(* IEC 61131-3 sources: std_i2980_v2.06_cp053/Source/IMM/ieccontrol/ODC1 (part 7) *)

         IF bGoToEndIf THEN
            aGoToEndIf(iColumn := i);
         ELSIF bGoToBeginLoop THEN
            bGoToBeginLoop := FALSE;
            aGoToBeginLoop(iColumn := i, iInstance := sv_ODCSequenceInt[i][iRow].iCount);
         ELSIF bGoToEndLoop THEN
            bGoToEndLoop := FALSE;
            aGoToEndLoop(iColumn := i, iInstance := sv_ODCSequenceInt[i][iRow].iCount);
         ELSE
            aIncreaseRow(iColumn := i, iEndRow := miEndRow);
         END_IF;
      END_IF;
   END_IF; //odcParallelInfo[i].bColumnActive
END_FOR;

//interesting for HMI to see state of the interpreter
sv_InterpreterParallelInfo := odcParallelInfo;

@END_Body

@@@BEG_Comment@@@
@TL(6)
Interpret the 2 dimensional ODC array.
(Responsible for auto cycle and combined movements)

This needs to be called cyclically until aStatus.bActive = FALSE
This can happen when the interpreter has reached the end of the array/sequence
or when a error happens during interpreting.
@@@END_Comment@@@

@BEG_Body
@TL(84)
(**************************************** WARNING ********************************************
 *** The KEBA Kemro K2 System including software is not intended for safety control tasks! ***
 ***                       For further information see Comment tab!                        ***
 *********************************************************************************************)

bFound := FALSE;
StepPos.iColumn := 0;
StepPos.iRow := 0;

FOR iTmpRow := SearchStartPos.iRow TO sv_iUsedRows DO

   IF iTmpRow = SearchStartPos.iRow THEN
      //start searching in the given column
      iSearchColumn := SearchStartPos.iColumn;
   ELSE
      //start searching in the first column
      iSearchColumn := 1;
   END_IF;

   FOR iTmpColumn := iSearchColumn TO sv_iUsedColumns DO
      IF sv_ODCSequence[iTmpColumn][iTmpRow].iCompId = DeviceId.CompId AND
         INT_TO_DINT(sv_ODCSequence[iTmpColumn][iTmpRow].iIndexId) = DeviceId.IndexId THEN
         IF sv_ODCSequence[iTmpColumn][iTmpRow].iMoveId = MoveId AND
            sv_ODCSequence[iTmpColumn][iTmpRow].iMoveDir = MoveDir AND
            (IntermediateCond = 0 OR // do not care about intermediate condion if we don't search for it?
                                     // FIXME check flag in MoveData instead??
             INT_TO_DINT(sv_ODCSequence[iTmpColumn][iTmpRow].iCount) = IntermediateCond) THEN
            fbDebugTrace2(nODCInterpreter, CONCAT('found exact match of MoveId ',
                                                  DINT_TO_STRING(DeviceId.CompId),
                                                  '.',
                                                  DINT_TO_STRING(DeviceId.IndexId),
                                                  ' ',
                                                  DINT_TO_STRING(MoveId),
                                                  '/',
                                                  DINT_TO_STRING(MoveDir),
                                                  ' ',
                                                  DINT_TO_STRING(IntermediateCond),
                                                  ' at pos:',
                                                  DINT_TO_STRING(iTmpRow),
                                                  '/',
                                                  DINT_TO_STRING(iTmpColumn)));

            StepPos.iColumn := iTmpColumn;
            StepPos.iRow := iTmpRow;
            bFound := TRUE;
            RETURN;

         ELSIF bAllowNonMatchingId AND sv_ODCSequence[iTmpColumn][iTmpRow].iMoveDir = MoveDir THEN
            fbDebugTrace2(nODCInterpreter, CONCAT('found NON exact match of MoveId ',
                                                  DINT_TO_STRING(DeviceId.CompId),
                                                  '.',
                                                  DINT_TO_STRING(DeviceId.IndexId),
                                                  ' ',
                                                  DINT_TO_STRING(MoveId),
                                                  '/',
                                                  DINT_TO_STRING(MoveDir),
                                                  ' ',
                                                  DINT_TO_STRING(IntermediateCond),
                                                  ' at pos:',
                                                  DINT_TO_STRING(iTmpRow),
                                                  '/',
                                                  DINT_TO_STRING(iTmpColumn)));
            StepPos.iColumn := iTmpColumn;
            StepPos.iRow := iTmpRow;
            bFound := TRUE;
         END_IF;
      END_IF;
   END_FOR;
END_FOR;

IF NOT bFound THEN
   fbDebugTrace2(nODCInterpreter, CONCAT('movement ',
                                          DINT_TO_STRING(DeviceId.CompId),
                                          '.',
                                          DINT_TO_STRING(DeviceId.IndexId),
                                          ' ',
                                          DINT_TO_STRING(MoveId),
                                          '/',
                                          DINT_TO_STRING(MoveDir),
                                          ' ',
                                          DINT_TO_STRING(IntermediateCond),
                                          ' not found in auto cycle'));
END_IF;

@END_Body

@@@BEG_Comment@@@
@TL(10)
Search a Movement in the ODC array by DeviceId, MoveId and MovedDir
and return the position in the array.

If bAllowNonMatchingId is TRUE only DeviceId and MoveDir need to match.
But it still tries to get the best match(MoveId equals)

If IntermediateCond is <> 0, it is also checked against iCount when checking for exact match.

When a movement is found bFound is TRUE and StepPos contains the position
of the movement in the ODC array
@@@END_Comment@@@

@BEG_Body
@TL(18)
(**************************************** WARNING ********************************************
 *** The KEBA Kemro K2 System including software is not intended for safety control tasks! ***
 ***                       For further information see Comment tab!                        ***
 *********************************************************************************************)

IF mbFatalError THEN
   mbFatalError := FALSE;

   (* unlock all movements locked by aStopInterpreterInternal *)
   DeviceIdAll.CompId := cCompAll;
   DeviceIdAll.IndexId := cAllDevIndex;

   fbLockUnlock(DeviceId := DeviceIdAll,
               MoveDir  := cMoveAll,
               MoveId   := cMoveAll,
               Mode     := nUnlock);
END_IF;

@END_Body

@@@BEG_Comment@@@
@TL(2)
Notify the Interpreter that the array has been reinitialized
(this clears the fatal error flag)
@@@END_Comment@@@

@BEG_Body
@TL(9)
(**************************************** WARNING ********************************************
 *** The KEBA Kemro K2 System including software is not intended for safety control tasks! ***
 ***                       For further information see Comment tab!                        ***
 *********************************************************************************************)

bError := mbFatalError OR mbNormalError;
bFinished := mbFinished;
bActive := mbActive;

@END_Body

@@@BEG_Comment@@@
@TL(1)
Actual status of the interpreter.
@@@END_Comment@@@

@BEG_Body
@TL(41)
(**************************************** WARNING ********************************************
 *** The KEBA Kemro K2 System including software is not intended for safety control tasks! ***
 ***                       For further information see Comment tab!                        ***
 *********************************************************************************************)

mbStepMode := TRUE;

//stop started movements
StartedMovements := sv_StartedManualMovements;
FOR i := 1 TO StartedMovements.iStartedMovements DO

   //get move number
   fbGetMoveNumber(DeviceId := StartedMovements.MoveData[i].DeviceId,
                   MoveId := StartedMovements.MoveData[i].MoveId,
                   MoveDir := StartedMovements.MoveData[i].MoveDir,
                   iMoveNumber => iMoveNr);

   IF NOT sv_MovementsAvailable[iMoveNr].pMovementData^.bFinishAtInterrupt THEN
      //stop movement
      fbStop(DeviceId := StartedMovements.MoveData[i].DeviceId);
   ELSE
      //movement should finish
      //increase number of active row because otherwise this movement is started
      //again when stepping fwd
      aIncreaseRow(iColumn := StartedMovements.MoveData[i].StepPos.iColumn,
                   iEndRow := miEndRow);
   END_IF;

END_FOR;

//disable steps
FOR i := 1 TO cMaxParallelMovements DO
   IF odcParallelInfo[i].bColumnActive THEN
      odcParallelInfo[i].bDisabled := TRUE;
   END_IF;
END_FOR;

mbActive := FALSE;

sv_InterpreterParallelInfo := odcParallelInfo;

@END_Body

@@@BEG_Comment@@@
@TL(0)

@@@END_Comment@@@

@BEG_Body
@TL(24)
(**************************************** WARNING ********************************************
 *** The KEBA Kemro K2 System including software is not intended for safety control tasks! ***
 ***                       For further information see Comment tab!                        ***
 *********************************************************************************************)

//reset relevant flags
FOR i := 1 TO cMaxParallelMovements DO
   IF odcParallelInfo[i].bColumnActive THEN
      odcParallelInfo[i].bStartSent := FALSE;
      odcParallelInfo[i].bStartConditionWarnPrinted := FALSE;
      odcParallelInfo[i].bActivatedChecked := FALSE;
      odcParallelInfo[i].bDisabled := FALSE;

      //set step state to "active"
      fbSetStepState.StepPos.iColumn := i;
      fbSetStepState.StepPos.iRow := odcParallelInfo[i].iRow;
      fbSetStepState(StepState := nStateActive);
   END_IF;

END_FOR;

mbActive := TRUE;
mbStepMode := FALSE;

@END_Body

@@@BEG_Comment@@@
@TL(0)

@@@END_Comment@@@

@BEG_Body
@TL(23)
(**************************************** WARNING ********************************************
 *** The KEBA Kemro K2 System including software is not intended for safety control tasks! ***
 ***                       For further information see Comment tab!                        ***
 *********************************************************************************************)

//enable steps
FOR i := 1 TO cMaxParallelMovements DO
   IF odcParallelInfo[i].bColumnActive THEN
      odcParallelInfo[i].bDisabled := FALSE;
      odcParallelInfo[i].bStartSent := FALSE;
      odcParallelInfo[i].bStartConditionWarnPrinted := FALSE;
      odcParallelInfo[i].bActivatedChecked := FALSE;

      //set step state to "active"
      fbSetStepState.StepPos.iColumn := i;
      fbSetStepState.StepPos.iRow := odcParallelInfo[i].iRow;
      fbSetStepState(StepState := nStateActive);
   END_IF;

END_FOR;

mbActive := TRUE;

@END_Body

@@@BEG_Comment@@@
@TL(0)

@@@END_Comment@@@

@BEG_Body
@TL(7)
(**************************************** WARNING ********************************************
 *** The KEBA Kemro K2 System including software is not intended for safety control tasks! ***
 ***                       For further information see Comment tab!                        ***
 *********************************************************************************************)

mbStepMode := FALSE;

@END_Body

@@@BEG_Comment@@@
@TL(0)

@@@END_Comment@@@

@BEG_Body
@TL(144)
(**************************************** WARNING ********************************************
 *** The KEBA Kemro K2 System including software is not intended for safety control tasks! ***
 ***                       For further information see Comment tab!                        ***
 *********************************************************************************************)

IF bStartInActualLine THEN
   iStartRow := odcParallelInfo[iColumn].iRow;
ELSE
   iStartRow := (odcParallelInfo[iColumn].iRow - 1);
END_IF;

//reset step state of actually active step
fbSetStepState.StepPos.iColumn := iColumn;
fbSetStepState.StepPos.iRow := odcParallelInfo[iColumn].iRow;
fbSetStepState(StepState := nStateDefault);

iNewActivatedColumn := 0;

//get next line with a "real" movement
FOR iTmpLine := iStartRow TO iEndRow BY -1 DO
   fbDebugTrace2(nODCInterpreter, CONCAT('decreasing IP of column ', DINT_TO_STRING(iColumn),
                                         ' to ', DINT_TO_STRING(iTmpLine)));

   iMoveId := sv_ODCSequence[iColumn][iTmpLine].iMoveId;

   IF (iMoveId = cMoveEndIf) THEN
      // end_if => check if this "if" instance is active or already completely executed
      iCount := sv_ODCSequence[iColumn][iTmpLine].iCount;
      IF (mIFConditionHelpData[iCount].iInternalCount < 2) THEN
         //if or else tree is active
         //set active line in this column to begin of this "if" or "else"
         //so that stepping bwd can continue before this "if / else"
         FOR iLine := (iTmpLine - 1) TO 1 BY -1 DO
            IF ((sv_ODCSequence[iColumn][iLine].iMoveId = cMoveIf) OR (sv_ODCSequence[iColumn][iLine].iMoveId = cMoveElse)) AND
               (sv_ODCSequence[iColumn][iLine].iCount = iCount) THEN
               odcParallelInfo[iColumn].iRow := (iLine - 1);  //set row to "start parallel" step
               EXIT;
            END_IF;
         END_FOR;
         mIFConditionHelpData[iCount].iInternalCount := (mIFConditionHelpData[iCount].iInternalCount - 1);
      ELSE
         //condition completely executed -> do not allow stepping into
         odcParallelInfo[iColumn].iRow := (iTmpLine + 1); //set row to "end parallel" step
         odcParallelInfo[iColumn].bDisabled := TRUE;
         SET_ALARM(Name := erNoStepBwdIntoCondition);
      END_IF;

      EXIT;
   ELSIF (iMoveId = cMoveEndLoop) THEN
      // end loop => stop stepping bwd here
      odcParallelInfo[iColumn].iRow := iTmpLine; //set row to "end loop" step
      odcParallelInfo[iColumn].bDisabled := TRUE;
      SET_ALARM(Name := erNoStepBwdIntoLoop);
      EXIT;
   ELSIF (iMoveId = cMoveBeginLoop) THEN
      // begin of loop => stop stepping bwd here (do not modify line number)
      odcParallelInfo[iColumn].bDisabled := TRUE;
      SET_ALARM(Name := erNoStepBwdOutOfLoop);
      EXIT;
   ELSIF (iMoveId = cMoveBeginSequence) OR (iMoveId = cMoveEndSequence) THEN
      ; // begin or end sequence
   ELSIF (iMoveId = cMoveNone) OR (iMoveId = cMoveBeginGroup) OR (iMoveId = cMoveEndGroup) THEN
      ; //empty step or begin group / end group
   ELSIF (iMoveId = cMoveIf) OR (iMoveId = cMoveElse) THEN
      ; //if , else
   ELSIF iMoveId = cMoveEndParallelOpen THEN
      ; //no special action necessary
   ELSIF iMoveId = cMoveEndParallel THEN
      //get according column and activate it
      FOR iTmpColumn := (iColumn + 1) TO sv_iUsedColumns DO
         IF sv_ODCSequence[iTmpColumn][iTmpLine].iMoveId = cMoveEndParallel THEN
            odcParallelInfo[iTmpColumn].bColumnActive := TRUE;
            odcParallelInfo[iTmpColumn].iRow := (iTmpLine + 1); //necessary to handle more end parallel in one line
            odcParallelInfo[iTmpColumn].bDisabled := TRUE;
            iNewActivatedColumn := iTmpColumn;
            EXIT;
         END_IF;
      END_FOR;
   ELSIF (iMoveId = cMoveStartParallel) OR (iMoveId = cMoveStartParallelOpen) THEN
      bContinueDecreasing := FALSE;
      FOR iTmpColumn := 1 TO sv_iUsedColumns DO
         IF (sv_ODCSequence[iTmpColumn][iTmpLine].iMoveId = cMoveStartParallel) OR
            (sv_ODCSequence[iTmpColumn][iTmpLine].iMoveId = cMoveStartParallelOpen) THEN

            //start parallel or start parallel open found
            IF iTmpColumn < iColumn THEN
               //SP left to actual column found
               //-> deactivate actual column and set line number
               odcParallelInfo[iColumn].iRow := iTmpLine;
               odcParallelInfo[iColumn].bDisabled := FALSE;
               odcParallelInfo[iColumn].bColumnActive := FALSE;
               IF sv_TraceLevel.bODCInterpreter THEN
                  dummy := Print('aDecreaseRow: deactivate column %d ',iColumn);
               END_IF;
            ELSE
               //SP is the most left one in this line
               //-> all SP to the right must be deactivated and their active row must be equal
               bOk := TRUE;
               FOR x := (iTmpColumn + 1) TO sv_iUsedColumns DO
                  //only consider SP entries
                  IF (sv_ODCSequence[x][iTmpLine].iMoveId = cMoveStartParallel) OR
                     (sv_ODCSequence[x][iTmpLine].iMoveId = cMoveStartParallelOpen) THEN
                     bParallelTreeReady := NOT odcParallelInfo[x].bColumnActive AND (odcParallelInfo[x].iRow = iTmpLine);
                     bOk := bOk AND bParallelTreeReady;
                  END_IF;
               END_FOR;

               IF bOk THEN
                  //all parallel trees ready -> decrease line of this column so that it can continue
                  bContinueDecreasing := TRUE;
               ELSE
                  //column still active -> wait in this line
                  odcParallelInfo[iColumn].iRow := iTmpLine;
                  odcParallelInfo[iColumn].bDisabled := TRUE;
                  bContinueDecreasing := FALSE;
               END_IF;
            END_IF;

            EXIT; //exit inner loop
         END_IF;
      END_FOR;

      IF NOT bContinueDecreasing THEN
         EXIT;  // exit outer loop
      END_IF;
   ELSE
      //valid step found -> set line number and disable this step
      IF sv_TraceLevel.bODCInterpreter THEN
         dummy := Print('///////// set active row of column %d to %d ////////////',iColumn, iTmpLine);
      END_IF;
      odcParallelInfo[iColumn].iRow := iTmpLine;
      odcParallelInfo[iColumn].bDisabled := TRUE;
      EXIT;
   END_IF;
END_FOR;

odcParallelInfo[iColumn].bStartSent := FALSE;
odcParallelInfo[iColumn].bStartConditionWarnPrinted := FALSE;
odcParallelInfo[iColumn].bActivatedChecked := FALSE;
odcParallelInfo[iColumn].bPosReachedArrayLinked := FALSE;
odcParallelInfo[iColumn].bMovementReadyArrayLinked := FALSE;

sv_InterpreterParallelInfo[iColumn] := odcParallelInfo[iColumn];

@END_Body

@@@BEG_Comment@@@
@TL(0)

@@@END_Comment@@@
@END_Body

@END_Contents
@@@BEG_Password@@@
NGhzZm9kYzQ=
@@@END_Password@@@

(* ---- ABLogger.pu ---- *)
(*
@h    ! WARNING !
@h    The Kemro K2 system (including software) only meets category B according to EN 954-1,
@h    thus it is not intended for usage in safety-relevant control applications in the field
@h    of personal safety (e.g. emergency stop).
@h    To implement potentially necessary safety-relevant control tasks, always use additional
@h    external safety devices that are intended for the particular purpose, and meet the necessary
@h    functional safety.
@h    For further information see EN 954-1 (EN ISO 13849-1) and/or the K2-x00 user manual, chapter
@h    "CE conformity, directives and standards".

algorithm block for debug purpose, can be used to log single trace lines to file
*)

IMPORT_OVER_LISTFILE
 KFILE_Open_Data
, KFILE_Status

END_IMPORT

ALGORITHM_BLOCK ABLogger #DUMMY_EDIT_BLOCK

VAR
 iResult : DINT (* transferred bytes, return value of KFILE_Read/Write *);
 sTraceString : STRING(255) (* local output trace string *);
END_VAR

ALGORITHM aWriteLine

VAR_INPUT
 sFileName : STRING(255) (* absolute file path *);
 bAppend : BOOL (* append log file *);
END_VAR

VAR_IN_OUT
 sText : STRING(255) (* trace string to log *);
END_VAR

VAR_TEMP
 FileOpenData : KFILE_Open_Data (* file open information *);
 FileStatus : KFILE_Status (* file state *);
 sNewline : STRING(2) := '$n';
 iLen : DINT;
END_VAR
#BEGIN_EDIT_BLOCK
IF (bAppend) THEN
   FileOpenData := KFILE_Open(Name := sFileName,
                              Mode := KFILE_Mode_AppendCreate);
ELSE
   FileOpenData := KFILE_Open(Name := sFileName,
                              Mode := KFILE_Mode_ReadWriteDelete);
END_IF;

IF (FileOpenData.Status = KFILE_Status_OK) THEN
   iLen := LEN(sText);
   IF iLen > 0 THEN
      // write data
      iResult := KFILE_Write(Token := FileOpenData.Token,
                             Length := iLen,
                             Buffer := sText);
   END_IF;
   // CR/LF
   iResult := KFILE_Write(Token := FileOpenData.Token,
                        Length := 2,
                        Buffer := sNewline);

   // close file
   FileStatus := KFILE_Close(Token := FileOpenData.Token);
ELSE
   sTraceString := CONCAT('Log to file failed - file ',  sFileName,
                           'possibly already opened!');

   (* @TODO ABDebugTrace... *)
END_IF;

;#END_EDIT_BLOCK END_ALGORITHM

ALGORITHM aWriteString

VAR_INPUT
 sFileName : STRING(255) (* absolute file path *);
 bAppend : BOOL (* append log file *);
END_VAR

VAR_IN_OUT
 sText : STRING(255) (* trace string to log *);
END_VAR

VAR_TEMP
 FileOpenData : KFILE_Open_Data (* file open information *);
 FileStatus : KFILE_Status (* file state *);
 iLen : DINT;
END_VAR
#BEGIN_EDIT_BLOCK
IF (bAppend) THEN
   FileOpenData := KFILE_Open(Name := sFileName,
                              Mode := KFILE_Mode_AppendCreate);
ELSE
   FileOpenData := KFILE_Open(Name := sFileName,
                              Mode := KFILE_Mode_ReadWriteDelete);
END_IF;

IF (FileOpenData.Status = KFILE_Status_OK) THEN
   iLen := LEN(sText);
   IF iLen > 0 THEN
      // write data
      iResult := KFILE_Write(Token := FileOpenData.Token,
                             Length := iLen,
                             Buffer := sText);
   END_IF;
   // close file
   FileStatus := KFILE_Close(Token := FileOpenData.Token);
ELSE
   sTraceString := CONCAT('Log to file failed - file ',  sFileName,
                          'possibly already opened!');

   (* @TODO ABDebugTrace... *)
END_IF;

;#END_EDIT_BLOCK END_ALGORITHM

END_ALGORITHM_BLOCK

#END_OF_IEC_PART

@Puma @IecEditor 6 95 @Pou 25
@@@BEG_Comment@@@
@h    ! WARNING !
@h    The Kemro K2 system (including software) only meets category B according to EN 954-1,
@h    thus it is not intended for usage in safety-relevant control applications in the field
@h    of personal safety (e.g. emergency stop).
@h    To implement potentially necessary safety-relevant control tasks, always use additional
@h    external safety devices that are intended for the particular purpose, and meet the necessary
@h    functional safety.
@h    For further information see EN 954-1 (EN ISO 13849-1) and/or the K2-x00 user manual, chapter
@h    "CE conformity, directives and standards".

algorithm block for debug purpose, can be used to log single trace lines to file
@@@END_Comment@@@

@BEG_Contents

@BEG_Func
@RT(17)FuncTreeContainer
0
@END_Func

@BEG_Const
@RT(18)ConstTreeContainer
0
@END_Const

@BEG_Export

@BEG_Kind
@ALGORITHM_BLOCK @RT(8)ABLogger @STRUCTURED_TEXT
@RT(0) @RT(0) @RT(0)
@END_Kind

@BEG_Dcl
@RT(16)DclTreeContainer
2
@Var @RT(7)iResult @RT(0) @T @F @DT @RT(4)DINT @RT(0) @T @T @BASIC 0 @F
@F @F
@T
@BEG_Attrib
3 @RT(0) @RT(51)transferred bytes, return value of KFILE_Read/Write @RT(0)
@END_Attrib
1 0 @F @F @F @F

@Var @RT(12)sTraceString @RT(0) @T @F @DT @RT(11)STRING(255) @RT(0) @T @T @STRING 0 @F @RT(3)255 @F
@F @F
@T
@BEG_Attrib
3 @RT(0) @RT(25)local output trace string @RT(0)
@END_Attrib
1 0 @F @F @F @F

@END_Dcl

@END_Export

@BEG_Body

2

@BEG_Export

@BEG_Algo
@ALGORITHM @RT(10)aWriteLine @STRUCTURED_TEXT
@RT(0) @RT(0) @RT(0) @F @F
@END_Algo

@BEG_Dcl
@RT(16)DclTreeContainer
7
@Var @RT(9)sFileName @RT(0) @T @F @DT @RT(11)STRING(255) @RT(0) @T @T @STRING 0 @F @RT(3)255 @F
@F @F
@T
@BEG_Attrib
3 @RT(0) @RT(18)absolute file path @RT(0)
@END_Attrib
1 1 @F @F @F @F

@Var @RT(7)bAppend @RT(0) @T @F @DT @RT(4)BOOL @RT(0) @T @T @BASIC 0 @F
@F @F
@T
@BEG_Attrib
3 @RT(0) @RT(15)append log file @RT(0)
@END_Attrib
1 1 @F @F @F @F

@Var @RT(5)sText @RT(0) @T @F @DT @RT(11)STRING(255) @RT(0) @T @T @STRING 0 @F @RT(3)255 @F
@F @F
@T
@BEG_Attrib
3 @RT(0) @RT(19)trace string to log @RT(0)
@END_Attrib
1 2 @F @F @F @F

@Var @RT(12)FileOpenData @RT(0) @T @T @DERIVED 0 @T @T @DT @RT(15)KFILE_Open_Data @RT(0) @T @T @UNKNOWN 0 @F
@F @F
@T
@BEG_Attrib
3 @RT(0) @RT(21)file open information @RT(0)
@END_Attrib
1 4 @F @F @F @F

@Var @RT(10)FileStatus @RT(0) @T @T @DERIVED 0 @T @T @DT @RT(12)KFILE_Status @RT(0) @T @T @UNKNOWN 0 @F
@F @F
@T
@BEG_Attrib
3 @RT(0) @RT(10)file state @RT(0)
@END_Attrib
1 4 @F @F @F @F

@Var @RT(8)sNewline @RT(0) @T @F @DT @RT(9)STRING(2) @RT(0) @T @T @STRING 0 @F @RT(1)2 @F
@F @F
@T
@BEG_Attrib
3 @RT(4)'$n' @RT(0) @RT(0)
@END_Attrib
1 4 @F @F @F @F

@Var @RT(4)iLen @RT(0) @T @F @DT @RT(4)DINT @RT(0) @T @T @BASIC 0 @F
@F @F
@T
@BEG_Attrib
3 @RT(0) @RT(0) @RT(0)
@END_Attrib
1 4 @F @F @F @F

@END_Dcl

@END_Export

@BEG_Export

@BEG_Algo
@ALGORITHM @RT(12)aWriteString @STRUCTURED_TEXT
@RT(0) @RT(0) @RT(0) @F @F
@END_Algo

@BEG_Dcl
@RT(16)DclTreeContainer
6
@Var @RT(9)sFileName @RT(0) @T @F @DT @RT(11)STRING(255) @RT(0) @T @T @STRING 0 @F @RT(3)255 @F
@F @F
@T
@BEG_Attrib
3 @RT(0) @RT(18)absolute file path @RT(0)
@END_Attrib
1 1 @F @F @F @F

@Var @RT(7)bAppend @RT(0) @T @F @DT @RT(4)BOOL @RT(0) @T @T @BASIC 0 @F
@F @F
@T
@BEG_Attrib
3 @RT(0) @RT(15)append log file @RT(0)
@END_Attrib
1 1 @F @F @F @F

@Var @RT(5)sText @RT(0) @T @F @DT @RT(11)STRING(255) @RT(0) @T @T @STRING 0 @F @RT(3)255 @F
@F @F
@T
@BEG_Attrib
3 @RT(0) @RT(19)trace string to log @RT(0)
@END_Attrib
1 2 @F @F @F @F

@Var @RT(12)FileOpenData @RT(0) @T @T @DERIVED 0 @T @T @DT @RT(15)KFILE_Open_Data @RT(0) @T @T @UNKNOWN 0 @F
@F @F
@T
@BEG_Attrib
3 @RT(0) @RT(21)file open information @RT(0)
@END_Attrib
1 4 @F @F @F @F

@Var @RT(10)FileStatus @RT(0) @T @T @DERIVED 0 @T @T @DT @RT(12)KFILE_Status @RT(0) @T @T @UNKNOWN 0 @F
@F @F
@T
@BEG_Attrib
3 @RT(0) @RT(10)file state @RT(0)
@END_Attrib
1 4 @F @F @F @F

@Var @RT(4)iLen @RT(0) @T @F @DT @RT(4)DINT @RT(0) @T @T @BASIC 0 @F
@F @F
@T
@BEG_Attrib
3 @RT(0) @RT(0) @RT(0)
@END_Attrib
1 4 @F @F @F @F

@END_Dcl

@END_Export

@BEG_Body
@TL(31)
IF (bAppend) THEN
   FileOpenData := KFILE_Open(Name := sFileName,
                              Mode := KFILE_Mode_AppendCreate);
ELSE
   FileOpenData := KFILE_Open(Name := sFileName,
                              Mode := KFILE_Mode_ReadWriteDelete);
END_IF;

IF (FileOpenData.Status = KFILE_Status_OK) THEN
   iLen := LEN(sText);
   IF iLen > 0 THEN
      // write data
      iResult := KFILE_Write(Token := FileOpenData.Token,
                             Length := iLen,
                             Buffer := sText);
   END_IF;
   // CR/LF
   iResult := KFILE_Write(Token := FileOpenData.Token,
                        Length := 2,
                        Buffer := sNewline);

   // close file
   FileStatus := KFILE_Close(Token := FileOpenData.Token);
ELSE
   sTraceString := CONCAT('Log to file failed - file ',  sFileName,
                           'possibly already opened!');

   (* @TODO ABDebugTrace... *)
END_IF;

@END_Body

@@@BEG_Comment@@@
@TL(0)

@@@END_Comment@@@

@BEG_Body
@TL(26)
IF (bAppend) THEN
   FileOpenData := KFILE_Open(Name := sFileName,
                              Mode := KFILE_Mode_AppendCreate);
ELSE
   FileOpenData := KFILE_Open(Name := sFileName,
                              Mode := KFILE_Mode_ReadWriteDelete);
END_IF;

IF (FileOpenData.Status = KFILE_Status_OK) THEN
   iLen := LEN(sText);
   IF iLen > 0 THEN
      // write data
      iResult := KFILE_Write(Token := FileOpenData.Token,
                             Length := iLen,
                             Buffer := sText);
   END_IF;
   // close file
   FileStatus := KFILE_Close(Token := FileOpenData.Token);
ELSE
   sTraceString := CONCAT('Log to file failed - file ',  sFileName,
                          'possibly already opened!');

   (* @TODO ABDebugTrace... *)
END_IF;

@END_Body

@@@BEG_Comment@@@
@TL(0)

@@@END_Comment@@@
@END_Body

@END_Contents
@@@BEG_Password@@@
NGhzZm9kYzQ=
@@@END_Password@@@
